(* Test scenarios for formal verification *)

(* Test 1: Humidity below 30% - should eventually turn on sprinklers *)
TestMoisture := 25.0;
WateringSystem(SoilMoistureSensor := TestMoisture, ResponseDelay := TestDelay);
@Assert(WateringSystem.SprinklersOn OR (WateringSystem.TargetSprinklerState AND NOT WateringSystem.DelayTimer.Q));

(* Test 2: Humidity above 70% - should eventually turn off sprinklers *)
TestMoisture := 75.0;
WateringSystem(SoilMoistureSensor := TestMoisture, ResponseDelay := TestDelay);
@Assert(NOT WateringSystem.SprinklersOn OR (NOT WateringSystem.TargetSprinklerState AND NOT WateringSystem.DelayTimer.Q));

(* Test 3: Humidity within hysteresis band - should maintain state *)
TestMoisture := 50.0;
WateringSystem(SoilMoistureSensor := TestMoisture, ResponseDelay := TestDelay);
@Assert(WateringSystem.TargetSprinklerState = WateringSystem.SprinklersOn);

(* Test 4: Input validation - ensure moisture is clamped to 0-100% *)
TestMoisture := -10.0;
WateringSystem(SoilMoistureSensor := TestMoisture, ResponseDelay := TestDelay);
@Assert(WateringSystem.ValidatedMoisture = 0.0);

TestMoisture := 110.0;
WateringSystem(SoilMoistureSensor := TestMoisture, ResponseDelay := TestDelay);
@Assert(WateringSystem.ValidatedMoisture = 100.0);

(* Test 5: Reachability - sprinklers can be turned on *)
@Assert(EXISTS TRUE : WateringSystem.SprinklersOn = TRUE);

(* Test 6: Reachability - sprinklers can be turned off *)
@Assert(EXISTS TRUE : WateringSystem.SprinklersOn = FALSE);
